{attribute 'GeneratedUsingTerminal: EL1382-0000-0016'}
{attribute addProperty BoxType "EL1382-0000-0016"}
{attribute addProperty Id "EtcSlaveTerminalBaseChannel_1AT %I*Channel_31CEFA7F2Channel_2AT %I*Channel_31CEFA7F2WcStateAT %I*WcState_9091E0EB2InfoDataAT %I*InfoData_6F19DB2B2"}
{attribute addProperty CRC "4266454968"}
{attribute addProperty Size "8"}
TYPE EL1382_FE4CEFB8 EXTENDS EtcSlaveTerminalBase :
STRUCT
	{attribute addProperty Name "Channel_1"}
	Channel_1 : Channel_31CEFA7F;
	{attribute addProperty Name "Channel_2"}
	Channel_2 : Channel_31CEFA7F;
	{attribute addProperty Name "WcState"}
	WcState : WcState_9091E0EB;
	{attribute addProperty Name "InfoData"}
	InfoData : InfoData_6F19DB2B;
END_STRUCT
END_TYPE

(* stored: Version 1.2.0.0, ProductVersion 3.1.4024.9
   DUT EL1382_FE4CEFB8: Id {5da28a53-90dc-4528-be2d-a2b2a0bced58} *)
